# EPICS alarm handler configuration: caQtDM_UnitTests/tst_qtcontrols/fixtures/alh/macros.alhConfig
GROUP NULL $(P)GROUP
CHANNEL $(P)GROUP $(P)$(R):ch
CHANNEL $(P)GROUP $(UNDEF):ch
